Staubli VAL3: flagStatus.dtx

public num RosFlag
public num RobotFlag
public num ForceFlag
